(* CoDeSys 2.3 export: PROCESSVARIABLEGROUP_TS.EXP *)

(* Data type in Diag/ProcessValues *)
TYPE ProcessVariableGroup_ts :
STRUCT
	GroupName_as8			: STRING(32);
(*	GroupName_as8			: ARRAY [1..4] OF STRING(32);*)
	ProcessVariable_as	: ARRAY [1..8] OF ProcessVariable_ts;
END_STRUCT
END_TYPE
